TYPE _ST_SETTINGS_ :
STRUCT
END_STRUCT
END_TYPE

(* stored: Version 1.1.0.1, ProductVersion 3.1.4022.18
   DUT _ST_SETTINGS_: Id {5ef149a8-5257-4e16-8d0c-d71d81e82caf} *)
